{attribute 'qualified_only'}
VAR_GLOBAL

	// general use I/O
	biOperatorDoorClosed 	AT %I* : BOOL;
	biMaintDoorClosed		AT %I* : BOOL;
	
	// stack light I/O
	boStackLightGreen		AT %Q* : BOOL;
	boStackLightYellow		AT %Q* : BOOL;
	boStackLightRed			AT %Q* : BOOL;
	
	// salt furnace I/O
	aiSaltTemp				AT %I* : INT;
	
	// quench tank I/O
	biWaterLevelLow			AT %I* : BOOL;
	biWaterLevelHigh 		AT %I* : BOOL;
	biWaterOverflowAlarm	AT %I* : BOOL;
	biWaterLeakAlarm		AT %I* : BOOL;
	boEnablePump			AT %Q* : BOOL;
	boOpenFillValve			AT %Q* : BOOL;
	boOpenDrainValve		AT %Q* : BOOL;
	boEnableHeaters			AT %Q* : BOOL;
	aiWaterTemp				AT %I* : USINT;
	
	// gantry I/O
	biMotorErrorX			AT %I* : BOOL;
	biMotorErrorY			AT %I* : BOOL;
	
END_VAR

(* stored: Version 1.1.0.1, ProductVersion 3.1.4024.11
   GVL GVL: Id {ea787d6c-627f-4fb6-88c4-d6ea0572f3b1} *)
